{attribute 'GeneratedUsingTerminal: EL9250--0000'}
{attribute addProperty BoxType "EL9250--0000"}
{attribute addProperty Description "EL9150 Power Supplier with LED(230V, Fuse)"}
{attribute addProperty Physics "KK"}
{attribute addProperty Id "EL9250"}
{attribute addProperty CRC "2483640354"}
{attribute addProperty Size "0"}
TYPE EL9250_94095822 EXTENDS EtcSlaveTerminalBase_947E5A46 :
STRUCT
END_STRUCT
END_TYPE

(* stored: Version 1.2.0.0, ProductVersion 3.1.4024.11
   DUT EL9250_94095822: Id {4c3ee9d8-f72b-40f0-9ea6-94f55dc90eb0} *)
